TYPE ST_ThNTZ_Parameter :
STRUCT
	Temp_Max				: REAL;
	Temp_Min				: REAL;
	Regelung_PI_Oben_Kp	: REAL;
	Regelung_PI_Oben_Tn	: DINT;
	Regelung_PI_Oben_Tctr	: DINT;

	Regelung_Sollw_KRITIKAL_OBEN_TEMP    : REAL;
	Regelung_Sollw_KRITIKAL_UNTEN_TEMP   : REAL;
	Regelung_Sollw_Max    : REAL;
	Regelung_Sollw_Min    : REAL;
	Regelung_Sollw_Max_Min : REAL;


	Stellwert_Leistung_Max		: REAL;
	Stellwert_Leistung_Min		: REAL;

	AutoQuittierung			: BOOL;



END_STRUCT
END_TYPE

(* stored: Version 1.1.0.1, ProductVersion 3.1.4024.9
   DUT ST_ThNTZ_Parameter: Id {8a12efdf-ef9c-4af2-854a-16a081f8b4bb} *)
